Universal Robots URScript: movej09.script

# movej:
# Set tcp: Use active tcp
# Joint speed : 60/s
# Joint acceleration : 80/s
# Use joint angles: none
# waypoint1: feature view, xyz-RxRyRz (radian), Joint positions (degree)
# stop at this point
# use shared parameters
# add until: expression digital_in[0]=1

def unnamed():
  global _hidden_verificationVariable=0
  step_count_e25e474f_e4af_4e37_87f0_5848f6533a25 = 0.0
  thread Step_Counter_Thread_ce51154b_e24e_4a1f_930a_358d9ddc85e2():
    while (True):
      step_count_e25e474f_e4af_4e37_87f0_5848f6533a25 = step_count_e25e474f_e4af_4e37_87f0_5848f6533a25 + 1.0
      sync()
    end
  end
  run Step_Counter_Thread_ce51154b_e24e_4a1f_930a_358d9ddc85e2()
  set_tcp(p[0.0,0.0,0.0,0.0,0.0,0.0])
  set_target_payload(1.000000, [0.000000, 0.000000, 0.000000], [0.001539, 0.001539, 0.001539, 0.000000, 0.000000, 0.000000])
  set_standard_analog_input_domain(0, 1)
  set_standard_analog_input_domain(1, 1)
  set_tool_analog_input_domain(0, 1)
  set_tool_analog_input_domain(1, 1)
  set_analog_outputdomain(0, 0)
  set_analog_outputdomain(1, 0)
  set_input_actions_to_default()
  set_tool_communication(False, 115200, 0, 1, 1.5, 3.5)
  set_tool_output_mode(0)
  set_tool_digital_output_mode(0, 1)
  set_tool_digital_output_mode(1, 1)
  set_tool_voltage(0)
  set_gravity([0.0, 0.0, 9.82])
  set_safety_mode_transition_hardness(1)
  global Waypoint_1_p=p[-.136861537556, -.267180821738, .146971261118, -.001221359682, 3.116276528482, .038891915637]
  global Waypoint_1_q=[-1.6006999999999998, -1.7271, -2.2029999999999994, -0.8079999999999998, 1.5951, -0.030999999999999694]
  while (True):
    $ 1 "Robot Program"
    $ 2 "MoveJ"
    $ 3 "Waypoint_1" "breakAfter"
    global move_thread_flag_3=0
    thread move_thread_3():
      enter_critical
      move_thread_flag_3 = 1
      movej(get_inverse_kin(Waypoint_1_p, qnear=Waypoint_1_q), a=1.3962634015954636, v=1.0471975511965976)
      move_thread_flag_3 = 2
      exit_critical
    end
    move_thread_flag_3 = 0
    move_thread_han_3 = run move_thread_3()
    while (True):
      if (get_standard_digital_in(0) == 1):
        kill move_thread_han_3
        stopj(1.3962634015954636)
        $ 4 "Until (expression)"
        break
      end
      sleep(1.0E-10)
      if (move_thread_flag_3 > 1):
        join move_thread_han_3
        break
      end
      sync()
    end
  end
end
